% RSLogix 500 project JSR.RSS, saved by version 8.30.00.15 %
PROJECT "UNTITLED"    % processor: MicroLogix 1400 %

PROGRAM FILES
  LAD 2   6 rungs
  LAD 3   4 rungs
  LAD 4   4 rungs

DATA FILES
  O0 OUTPUT  6 elements
  I1 INPUT  8 elements
  S2 STATUS  66 elements
  B3 BINARY  1 elements
  T4 TIMER  2 elements
  C5 COUNTER  1 elements
  R6 CONTROL  1 elements
  N7 INTEGER  1 elements
  F8 FLOAT  1 elements

LADDER 2
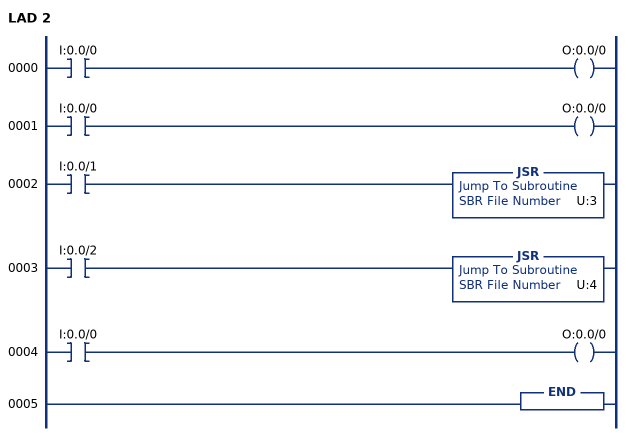
% Rung: 0 %
SOR XIC I:0.0/0 OTE O:0.0/0 EOR
% Rung: 1 %
SOR XIC I:0.0/0 OTE O:0.0/0 EOR
% Rung: 2 %
SOR XIC I:0.0/1 JSR U:3 EOR
% Rung: 3 %
SOR XIC I:0.0/2 JSR U:4 EOR
% Rung: 4 %
SOR XIC I:0.0/0 OTE O:0.0/0 EOR
% Rung: 5 %
SOR END EOR

LADDER 3
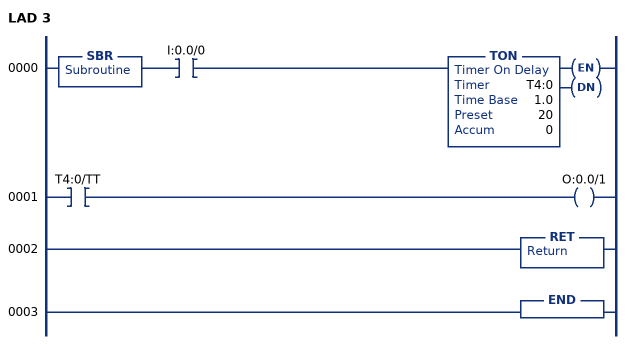
% Rung: 0 %
SOR SBR XIC I:0.0/0 TON T4:0 1.0 20 0 EOR
% Rung: 1 %
SOR XIC T4:0/TT OTE O:0.0/1 EOR
% Rung: 2 %
SOR RET EOR
% Rung: 3 %
SOR END EOR

LADDER 4
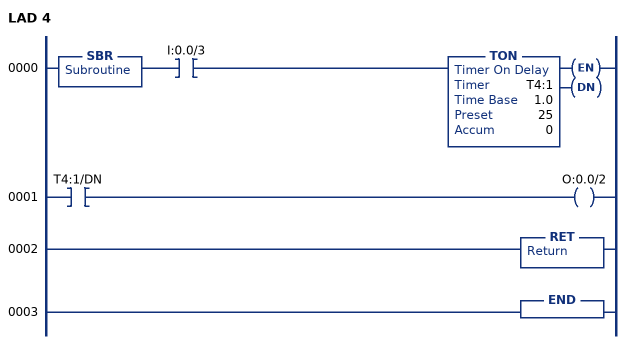
% Rung: 0 %
SOR SBR XIC I:0.0/3 TON T4:1 1.0 25 0 EOR
% Rung: 1 %
SOR XIC T4:1/DN OTE O:0.0/2 EOR
% Rung: 2 %
SOR RET EOR
% Rung: 3 %
SOR END EOR

DATA TABLE (non-zero values as saved)
DATA T4
% .PRE .ACC %
% T4:0 % 20 0
% T4:1 % 25 0
